(* PLC project Unnamed, Unknown Unnamed 1 *)
(* stored: creationDateTime 2019-06-12T10:21:38, modificationDateTime 2019-06-12T10:51:05 *)

PROGRAM wave_generator
  VAR
    oscilator : BOOL;
    count_up : BOOL;
    count_down : BOOL;
  END_VAR
  VAR
    output AT %QW0 : UINT;
  END_VAR
  VAR
    TON0 : TON;
    TOF0 : TOF;
    CTUD_UDINT0 : CTUD_UDINT;
  END_VAR
  VAR  (* added by the conversion: wires and edge detectors of the diagram *)
    _EQ9_OUT : BOOL;
    _EQ14_OUT : BOOL;
    R_TRIG1 : R_TRIG;
    R_TRIG2 : R_TRIG;
  END_VAR

(* LD diagram, written out as Structured Text *)
(* Main Oscilator - Used to generate the base frequency for the Up/Down Counter *)
TON0(IN := NOT oscilator, PT := T#100ms);
TOF0(IN := TON0.Q, PT := T#100ms);
oscilator := TOF0.Q;
(* Comparator testers. Used to switch the count from up/down and vice-versa *)
_EQ9_OUT := output = 0;
IF _EQ9_OUT THEN count_up := TRUE; END_IF;
IF _EQ9_OUT THEN count_down := FALSE; END_IF;
_EQ14_OUT := output = 100;
IF _EQ14_OUT THEN count_down := TRUE; END_IF;
IF _EQ14_OUT THEN count_up := FALSE; END_IF;
(* Main Up/Down Counter. The Current Value (CV) is the output we need *)
R_TRIG1(CLK := oscilator AND count_up);
R_TRIG2(CLK := oscilator AND count_down);
CTUD_UDINT0(CU := R_TRIG1.Q, CD := R_TRIG2.Q, PV := 65536);
output := UDINT_TO_UINT(CTUD_UDINT0.CV);
END_PROGRAM

CONFIGURATION Config0
  RESOURCE Res0 ON PLC
    TASK task0(INTERVAL := T#20ms, PRIORITY := 0);
    PROGRAM instance0 WITH task0 : wave_generator;
  END_RESOURCE
END_CONFIGURATION
